(* Logix 5000 project; controller EuniceF_ICA15 vendor 1 type 14 code 150 rev 37.11; software revision 37.00 *)

TASK MainTask (continuous, watchdog 500 ms) : MainProgram

MODULES
   Local : vendor 1 type 14 code 150 (Compact 0, rev 37.11)
      Discrete_IO : Embedded (Compact 1, rev 3.1, Output RPI 20 ms)
      Analog_IO : Embedded (Compact 2, rev 1.1, Output RPI 80 ms)
      Counters : Embedded (Compact 3, rev 1.1, Output RPI 20 ms)
END_MODULES

VAR_GLOBAL   (* controller tags *)
   Motor : ALIAS FOR Local:1:O.Data.1;
   seq1 : DINT;
   Switch : ALIAS FOR Local:1:I.Data.11;
END_VAR

PROGRAM MainProgram   (* main routine MainRoutine *)

ROUTINE MainRoutine   (* ladder *)
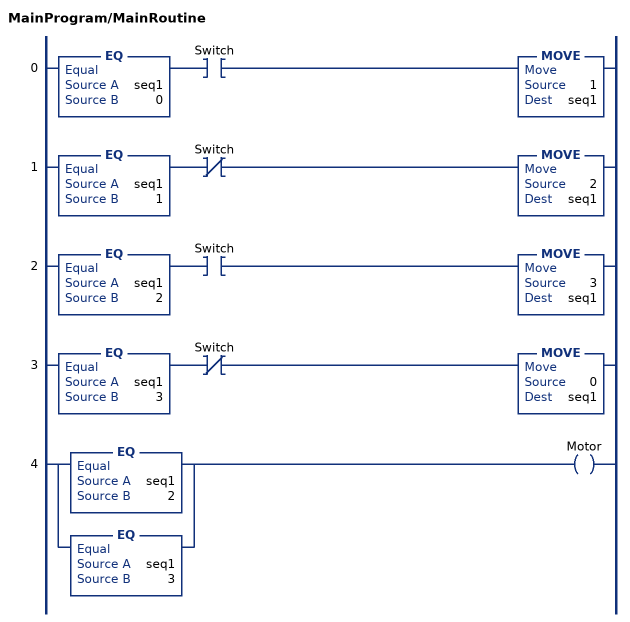
   0: EQ(seq1,0)XIC(Switch)MOVE(1,seq1);
   1: EQ(seq1,1)XIO(Switch)MOVE(2,seq1);
   2: EQ(seq1,2)XIC(Switch)MOVE(3,seq1);
   3: EQ(seq1,3)XIO(Switch)MOVE(0,seq1);
   4: [EQ(seq1,2) ,EQ(seq1,3) ]OTE(Motor);
END_ROUTINE
END_PROGRAM
